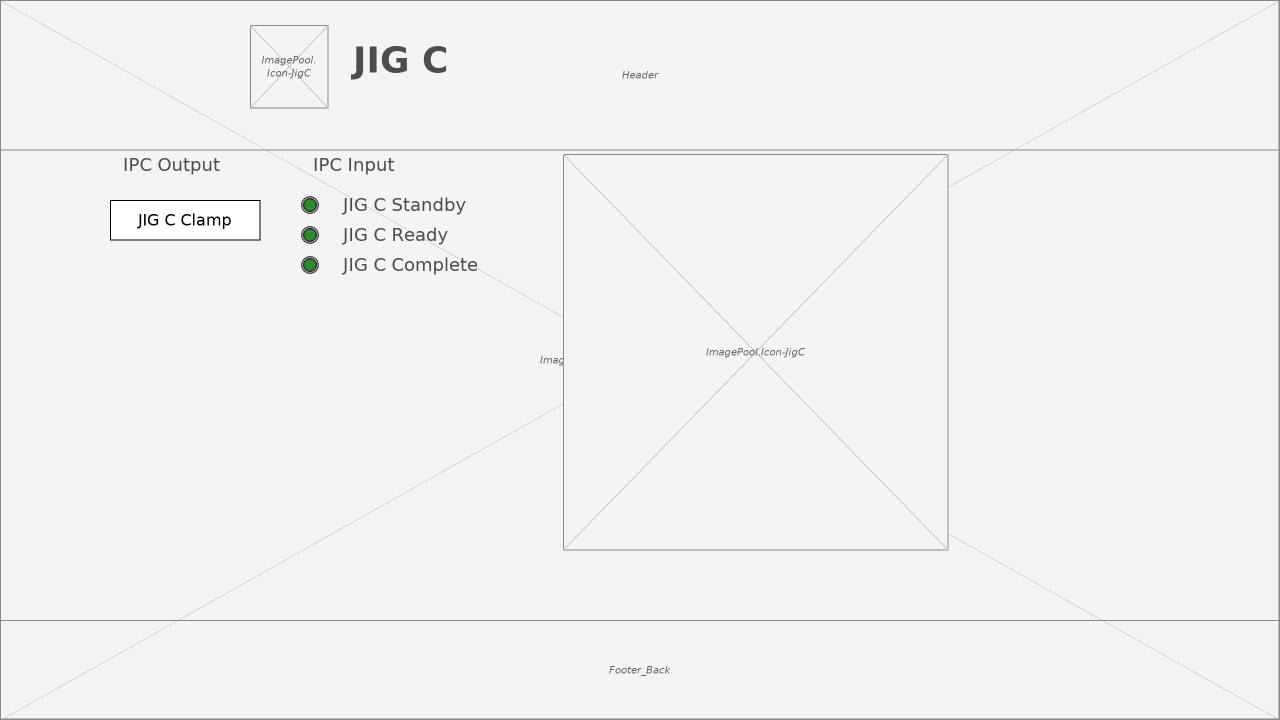
VISUALIZATION PAGE_JIG_C  // 1280x720
    Image (0,0 1280x720), image: ImagePool.The-New-Silver-Backgrounds
    Frame (0,620 1280x100)
        shows Footer_Back()
    Frame (0,0 1280x150)
        shows Header()
    Label (350,40 300x40), "JIG C"
    Label (120,150 150x30), "IPC Output"
    RoundedRectangle (110,200 150x40), "JIG C Clamp"
        toggle GVL.JIGC_Clamp
    Label (310,150 150x30), "IPC Input"
    Label (340,220 170x30), "JIG C Ready"
    Lamp1 (300,225 20x20), variable: GVL.JIGC_Ready, style: Lamp-Lamp1-Green
    Label (340,190 170x30), "JIG C Standby"
    Lamp1 (300,195 20x20), variable: GVL.JIGC_Standby, style: Lamp-Lamp1-Green
    Image (250,25 78x83), image: ImagePool.Icon-JigC
    Image (563,154 385x396), image: ImagePool.Icon-JigC
    Label (340,250 170x30), "JIG C Complete"
    Lamp1 (300,255 20x20), variable: GVL.JIGC_Complete, style: Lamp-Lamp1-Green
END_VISUALIZATION

(* stored: Version 1.1.0.1, ProductVersion 3.1.4024.12
   Visu PAGE_JIG_C: Id {10d41be6-2fc0-4086-9d6e-5a5129d17299} *)
